TYPE
    TcoFeeding_Status_v_1_x_x EXTENDS TcoCore.TcoStruct :
    STRUCT

	
		{attribute addProperty Name "<#Action#>"}
        ActionDescription : STRING;
		
		{attribute addProperty Name "<#Safety conditon met#>"}
        SafeCondition : BOOL;

    END_STRUCT
END_TYPE

(* stored: Version 1.1.0.1
   DUT TcoFeeding_Status_v_1_x_x: Id {dbdc34e1-3b9b-4743-9523-db185c563826} *)
